// TIA Portal V18 export
TYPE "Starter_HPU_IO_Out"
   STRUCT
      Slot2 { S7_SetPoint := 'True'} : "TM_Count_Man_Out";
      Slot7 { S7_SetPoint := 'True'} : "TM_Pulse_2x24_Out";
      Slot8 { S7_SetPoint := 'True'} : "TM_Pulse_2x24_Out";
      Slot9 { S7_SetPoint := 'True'} : "TM_Pulse_2x24_Out";
      Slot10 { S7_SetPoint := 'True'} : "RQ_4x120VDC/5A_In";
      Slot11 { S7_SetPoint := 'True'} : "RQ_4x120VDC/5A_In";
      Slot12 { S7_SetPoint := 'True'} : "RQ_4x120VDC/5A_In";
      Slot13 { S7_SetPoint := 'True'} : "RQ_4x120VDC/5A_In";
      Slot14 { S7_SetPoint := 'True'} : "RQ_4x120VDC/5A_In";
      Slot15 { S7_SetPoint := 'True'} : "RQ_4x120VDC/5A_In";
      Slot16 { S7_SetPoint := 'True'} : "RQ_4x120VDC/5A_In";
      Slot17 { S7_SetPoint := 'True'} : "RQ_4x120VDC/5A_In";
   END_STRUCT;
END_TYPE
